SUBAPPLICATION ManyOutputsSIFB050 (* Subapplication Type *)
  (* Standard: 61499-2 *)
  (* Version 1.0, 2025-05-03, cochicde *)
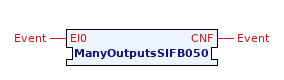
  EVENT_INPUT
    EI0;
  END_EVENT
  EVENT_OUTPUT
    CNF;
  END_EVENT
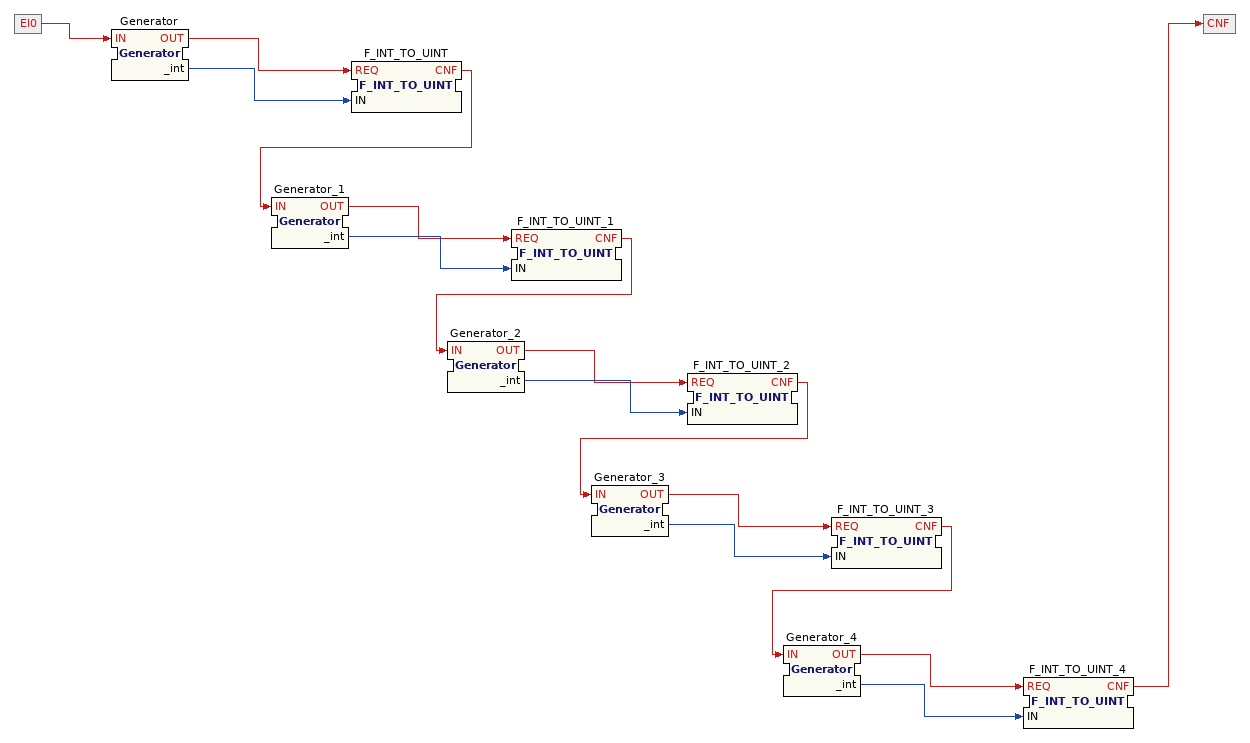
  FBS
    F_INT_TO_UINT_1 : F_INT_TO_UINT;
    Generator : performance::Generator;
    Generator_1 : performance::Generator;
    Generator_2 : performance::Generator;
    F_INT_TO_UINT_4 : F_INT_TO_UINT;
    F_INT_TO_UINT : F_INT_TO_UINT;
    Generator_3 : performance::Generator;
    F_INT_TO_UINT_2 : F_INT_TO_UINT;
    F_INT_TO_UINT_3 : F_INT_TO_UINT;
    Generator_4 : performance::Generator;
  END_FBS
  EVENT_CONNECTIONS
    Generator_1.OUT TO F_INT_TO_UINT_1.REQ;
    F_INT_TO_UINT_1.CNF TO Generator_2.IN;
    Generator.OUT TO F_INT_TO_UINT.REQ;
    F_INT_TO_UINT.CNF TO Generator_1.IN;
    Generator_2.OUT TO F_INT_TO_UINT_2.REQ;
    Generator_4.OUT TO F_INT_TO_UINT_4.REQ;
    F_INT_TO_UINT_2.CNF TO Generator_3.IN;
    Generator_3.OUT TO F_INT_TO_UINT_3.REQ;
    F_INT_TO_UINT_3.CNF TO Generator_4.IN;
    EI0 TO Generator.IN;
    F_INT_TO_UINT_4.CNF TO CNF;
  END_CONNECTIONS
  DATA_CONNECTIONS
    Generator_1._int TO F_INT_TO_UINT_1.IN;
    Generator._int TO F_INT_TO_UINT.IN;
    Generator_2._int TO F_INT_TO_UINT_2.IN;
    Generator_4._int TO F_INT_TO_UINT_4.IN;
    Generator_3._int TO F_INT_TO_UINT_3.IN;
  END_CONNECTIONS
END_SUBAPPLICATION
